INTERFACE I_Clock
// Interface for every time dependent method

PROPERTY milliseconds : ULINT
GET
END_GET
SET
END_SET
END_PROPERTY

PROPERTY nanoseconds : ULINT
GET
END_GET
SET
END_SET
END_PROPERTY

METHOD Run : BOOL
VAR_INPUT
END_VAR
END_METHOD

PROPERTY seconds : ULINT
GET
END_GET
SET
END_SET
END_PROPERTY

END_INTERFACE

(* stored: Version 1.1.0.1, ProductVersion 3.1.4024.6
   Itf I_Clock: Id {fe9741fb-f3cc-4c6d-9cd4-5dbd144a7176}
   Property milliseconds: Id {81a36bb7-ce70-49ea-bb69-9c7a2ea8f956}
   Get Get: Id {edf9b888-8270-4967-8499-4846d80a4b44}
   Set Set: Id {af9cf0f8-62bf-4f39-87dc-4ce5992010de}
   Property nanoseconds: Id {c87822df-d528-45b2-81a9-1f52f134750e}
   Get Get: Id {f0af0f42-6c71-4986-9143-79a5d0dae0ad}
   Set Set: Id {88e6d234-6ad5-4669-b88a-6d50db8d921f}
   Method Run: Id {31e97ae0-ae5a-46cd-b63b-0b5a265c6ca7}
   Property seconds: Id {9f0f52c9-6e21-41f4-a5db-e65044d420fc}
   Get Get: Id {dd16df9e-0349-4fe6-8f01-77ac9fd48209}
   Set Set: Id {ad919a90-3a2b-4032-9be4-2cd50af0bcc0} *)
